TEXTLIST TL_Params_INT
  1 = 'App_HmiType'
  2 = 'TermChannel'
  3 = 'ExtruderId'
  4 = 'ModuleId'
  5 = 'ZoneId'
  6 = 'SupplyId'
  7 = 'CJ_CompMode'
  8 = 'CJ_CompZone'
  9 = 'SensTermSwapIdx'
  10 = 'HeaterSwapIdx'
  11 = 'CoolerSwapIdx'
  12 = 'nPwmFactorC'
  13 = '*** not Used ***'
  14 = '*** not Used ***'
  15 = '*** not Used ***'
  16 = '*** not Used ***'
  17 = '*** not Used ***'
  18 = '*** not Used ***'
  19 = '*** not Used ***'
  20 = '*** not Used ***'
  21 = '*** not Used ***'
  22 = '*** not Used ***'
  23 = '*** not Used ***'
  24 = '*** not Used ***'
  25 = '*** not Used ***'
  26 = '*** not Used ***'
  27 = '*** not Used ***'
  28 = '*** not Used ***'
  29 = '*** not Used ***'
  30 = '*** not Used ***'
  31 = '*** not Used ***'
  32 = '*** not Used ***'
  33 = '*** not Used ***'
  34 = '*** not Used ***'
  35 = '*** not Used ***'
  36 = '*** not Used ***'
  37 = '*** not Used ***'
  38 = '*** not Used ***'
  39 = '*** not Used ***'
  40 = '*** not Used ***'
   = ''
END_TEXTLIST

(* stored: Version 1.1.0.1, ProductVersion 3.1.4018.5
   TextList TL_Params_INT: Id {d91a9f3d-45e7-4725-b4e2-f8f20bb06e63} *)
